FUNCTION_BLOCK RS_NoReset
//Output reset the input if the input is false 
VAR_INPUT
	Set 		: BOOL;
	Reset 		: BOOL;
END_VAR
VAR_OUTPUT
	Q1 			: BOOL;
END_VAR
VAR
	TRIG 		: R_TRIG;
	RS 			: RS;
END_VAR

TRIG(CLK := Set);
RS(Set := TRIG.Q, RESET1 := Reset AND NOT Set, Q1 => Q1);

END_FUNCTION_BLOCK

(* stored: Version 1.1.0.1, ProductVersion 3.1.4024.6
   POU RS_NoReset: Id {06d5e7d8-d88d-4ccf-8631-7aa2ef23dbe4}, SpecialFunc None *)
